{attribute 'qualified_only'}
{attribute 'strict'}
{attribute 'to_string'}
TYPE RollingFileState :
(
	Closed,
	Open,
	Writing,
	RollingOver
);
END_TYPE

(* stored: Version 1.1.0.1
   DUT RollingFileState: Id {418d9e79-3798-4452-9e4d-1876133876a3} *)
